Staubli VAL3: selectItem.pgx

public program selectItem(num x_nIndex (dimensions=1))
  local string l_sItem
  local TrajectoryItem l_tTraj
begin
  //
  // select or unselect one item
  //
  call trajType:getTrajItem(l_tTraj,x_nIndex)
  // check for the selected flag
  if find(l_tTraj.comment,"#")==-1
    l_tTraj.comment="#"+l_tTraj.comment
  else
    l_tTraj.comment=right(l_tTraj.comment,len(l_tTraj.comment)-1)
  endIf
  // set it
  call trajType:setTrajItem(l_tTraj,x_nIndex)
end
